{attribute 'linkalways'} 
{attribute 'no_explicit_call' := 'This FB is a CLASS and must be accessed using methods or properties'}
{attribute 'enable_dynamic_creation'}
FUNCTION_BLOCK Node_F_VN_KeyPointsGFTTExp EXTENDS VisionNode
VAR
    ipSrcImage : _ITcVnImage;
    ipKeyPoints : _ITcVnContainer;
    ipMask : _ITcVnImage;
    stParams : _TcVnParamsGFTT;
    hrPrev : _HRESULT(S_OK);
	hresult : _HRESULT(S_OK);
END_VAR

METHOD PUBLIC  Clone : I_Node
VAR
	pNode : POINTER TO Node_F_VN_KeyPointsGFTTExp;
END_VAR
pNode := __NEW(Node_F_VN_KeyPointsGFTTExp);
Clone := pNode^;
END_METHOD

METHOD FB_init : BOOL
VAR_INPUT
	bInitRetains : BOOL; // if TRUE, the retain variables are initialized (warm start / cold start)
	bInCopyCode : BOOL;  // if TRUE, the instance afterwards gets moved into the copy code (online change)
END_VAR
AddInput('ipSrcImage', ipSrcImage);
AddInput('ipMask', ipMask);
AddInput('stParams', stParams);
AddInput('hrPrev', hrPrev);
AddOutput('ipKeyPoints', ipKeyPoints);
AddOutput('hresult',hresult);
END_METHOD

METHOD PROTECTED OnExecute
hresult.Value := F_VN_KeyPointsGFTTExp(
	ipSrcImage := ipSrcImage.Value,
    ipKeyPoints := ipKeyPoints.Value,
    ipMask := ipMask.Value,
    stParams := stParams.Value,
	hrPrev:= hrPrev.Value);
END_METHOD

METHOD PUBLIC PreExecutionCheck
VAR_INPUT
	Check : I_PreExecutionChecks;
END_VAR
Check.IsTrue(ipSrcImage.IsValid, 'ipSrcImage must contain an image');
Check.IsTrue(ipSrcImage.HasChannelCount(1), 'ipSrcImage must have 1 channel');
END_METHOD

END_FUNCTION_BLOCK

(* stored: Version 1.1.0.1, ProductVersion 3.1.4024.15
   POU Node_F_VN_KeyPointsGFTTExp: Id {b99d062e-8397-029e-3e65-fad6eef494c8}, SpecialFunc None
   Folder Constructor: Id {eb6cf5ff-fd75-074a-02a0-5b7d7659d8a3}
   Method Clone: Id {60972a66-1c37-00b6-0c3c-719e7406b62f}
   Method FB_init: Id {14814c0f-dbd1-0a0e-39b6-d3551711c305}
   Method OnExecute: Id {6f7bc860-e688-0a81-132f-2be3881470e7}
   Method PreExecutionCheck: Id {3979e894-cfb3-0452-0b46-57c685c18814} *)
